Universal Robots PolyScope program: jenga_FIRE.urp

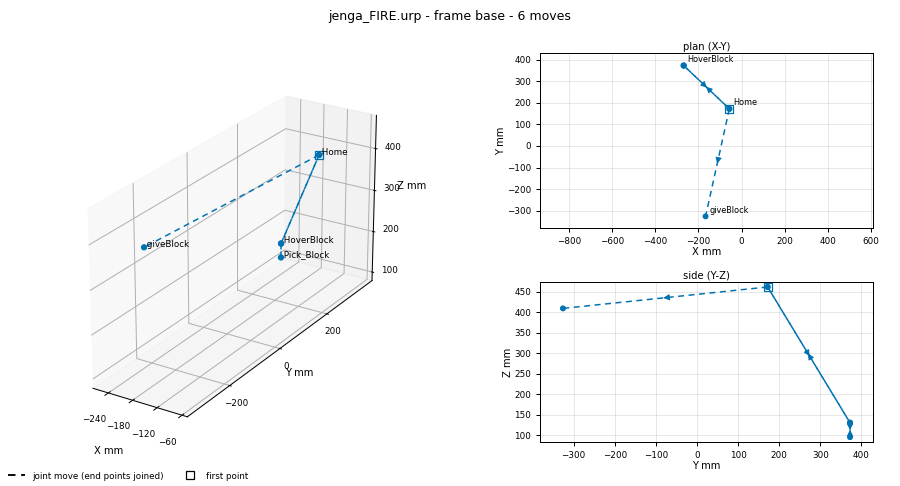
[picture p0: tool path of jenga_FIRE.urp in frame base, 6 of 6 moves have a stored position in this frame; points joined in program order, loops and branches not executed]
Program jenga_FIRE (installation=default directory=/programs/usbdisk createdIn=3.7.0.40195 lastSavedIn=3.15.8.106339 robotSerialNumber=2016330767)
Calibrated DH parameters: a=[-0.000074, -0.243398, -0.210699, 0.000027, 0.000052, 0]; d=[0.152002, 7.276382, 4.282012, -11.445796, 0.085202, 0.08239]; alpha=[1.566699, -0.002407, -0.002983, 1.569705, -1.570531, 0]; deltaTheta=[0.000021, -0.071916, -0.090359, 0.162183, -0.000005, -0.000082]
Robot Program (runOnlyOnce=false)
  MoveJ speed 60 deg/s, acceleration 80 deg/s^2 (useActiveTCP=true)
    Waypoint Home: TCP in base x=-57.158 y=171.878 z=461.129 mm, rx=-1.4823 ry=-0.8275 rz=0.756 rad; joints [-215.68, -51.594, -118.015, -14.484, 93.304, -360.754] deg
    Popup Message (haltProgram=false message=wait for block inputType=Text)
    MoveJ speed 60 deg/s, acceleration 80 deg/s^2 (useActiveTCP=true)
      Waypoint HoverBlock: TCP in base x=-268.501 y=372.263 z=131.073 mm, rx=2.8371 ry=1.3483 rz=0.0354 rad; joints [-219.846, -136.043, -74.065, -60.449, 88.827, -360.754] deg
      Wait Sleep waitTime=1
      Waypoint Pick_Block: TCP in base x=-268.607 y=372.343 z=95.845 mm, rx=-2.8367 ry=-1.3482 rz=-0.0354 rad; joints [-219.819, -140.779, -75.83, -53.908, 88.817, -360.754] deg
      Wait Sleep waitTime=1
      Waypoint HoverBlock: TCP in base x=-268.501 y=372.263 z=131.073 mm, rx=2.8371 ry=1.3483 rz=0.0354 rad; joints [-219.846, -136.043, -74.065, -60.449, 88.827, -360.754] deg
      Popup Message (haltProgram=false message=pickBlock inputType=Text)
    MoveJ speed 60 deg/s, acceleration 80 deg/s^2 (useActiveTCP=true)
      Waypoint Home: TCP in base x=-57.158 y=171.878 z=461.129 mm, rx=-1.4823 ry=-0.8275 rz=0.756 rad; joints [-215.68, -51.594, -118.015, -14.484, 93.304, -360.754] deg
      Popup Message (haltProgram=false message=wait for operator readiness inputType=Text)
    MoveJ speed 60 deg/s, acceleration 80 deg/s^2 (useActiveTCP=true)
      Waypoint giveBlock: TCP in base x=-167.206 y=-325.952 z=409.041 mm, rx=0.0928 ry=-3.0439 rz=0.0199 rad; joints [-98.296, -107.136, -43.927, -117.256, 84.724, -371.735] deg
      Popup Message (haltProgram=false message=wait for human operator to hold block inputType=Text)
